(* CODESYS project FsGenerics_0.1.1.1.library
   Company: FisoThemes
   DefaultNamespace: FsGenerics
   Version: 0.1.1.1
   Placeholder: FsGenerics
   Author: Goodwill Mzumala
   Description: A library for handling generic data.
   Title: FsGenerics

Project tree, tasks and I/O mapping:
  libraries: FsCommon, * (FisoThemes); FsError, * (FisoThemes); Tc2_Standard, * (Beckhoff Automation GmbH); Tc2_System, * (Beckhoff Automation GmbH); Tc2_Utilities, * (Beckhoff Automation GmbH); Tc3_Module, * (Beckhoff Automation GmbH)
  DUTs/
  GVLs/
  ITFs/
  PARAMs/
  POUs/
    function F_AllocateMemoryGeneric [ST]
    function F_AnyToGeneric [ST]
    function F_AnyToString [ST]
    function F_CloneGeneric [ST]
    function F_CompareAny [ST]
    function F_CompareGenerics [ST]
    function F_CopyGeneric [ST]
    function F_DeallocateGeneric [ST]
    function F_GenericToDateTime [ST]
    function F_GenericToNumber [ST]
    function F_GenericToString [ST]
    function F_GenericToTime [ST]
    function F_GenericToTimeOfDay [ST]
    function F_IsBooleanGeneric [ST]
    function F_IsDateGeneric [ST]
    function F_IsIntegerGeneric [ST]
    function F_IsMatchingGenerics [ST]
    function F_IsNumberGeneric [ST]
    function F_IsPrimitiveGeneric [ST]
    function F_IsRealNumberGeneric [ST]
    function F_IsSignedIntegerGeneric [ST]
    function F_IsStringConvertableGeneric [ST]
    function F_IsStringGeneric [ST]
    function F_IsTimeGeneric [ST]
    function F_IsUnsignedIntegerGeneric [ST]
    function F_ResetGeneric [ST]
    function F_SwapAny [ST]
    function F_SwapGenericsParameters [ST]
    program PLAYGROUND [ST]
  Project Information/
    function F_GetCompany [ST]
    function F_GetTitle [ST]
    function F_GetVersion [ST]
  UMLs/
  Version/
    global variables Global_Version
  VISUs/
*)

// Version/Global_Version
{attribute 'TcGenerated'}
{attribute 'no-analysis'}
{attribute 'linkalways'}
// This function has been automatically generated from the project information.
VAR_GLOBAL CONSTANT
	{attribute 'const_non_replaced'}
	stLibVersion_FsGenerics : ST_LibVersion := (iMajor := 0, iMinor := 1, iBuild := 1, iRevision := 1, nFlags := 0, sVersion := '0.1.1.1');
END_VAR

// POUs/F_AllocateMemoryGeneric
// Allocates memory for an array of generic values.
// [warning] This function performs dynamic memory allocation. Ensure proper error handling
//           and resource management to avoid memory leaks or allocation failures.
FUNCTION F_AllocateMemoryGeneric : POINTER TO FsCommon.T_Generic // Pointer to the allocated memory for generic values.
VAR_INPUT
	Count : FsCommon.T_Size; // The number of `FsCommon.T_Generic` values to allocate memory for.
END_VAR
VAR_OUTPUT
	Error : FsError.T_Error; // Error information if memory allocation fails.
END_VAR
VAR
	i, End : FsCommon.T_Position;
END_VAR

IF Count = 0 THEN RETURN; END_IF

F_AllocateMemoryGeneric := FsCommon.F_AllocateMemory(Count * SIZEOF(FsCommon.T_Generic));

IF F_AllocateMemoryGeneric = 0 THEN 
	Error := FsError.F_CreateError(
		FsError.GVL_ErrorDescriptors.fbGeneralErrorCodes,
		FsError.E_GeneralErrorCode.ERR_MEMORY_ALLOCATION_FAILED);
	RETURN;
	END_IF

End := FsCommon.F_SizeToPosition(Count) - 1;
FOR i := 0 TO End DO
	F_AllocateMemoryGeneric[i].TypeClass := __SYSTEM.TYPE_CLASS.TYPE_NONE;
	END_FOR

END_FUNCTION

// POUs/F_AnyToGeneric
// Converts a value of any type to a generic type.
FUNCTION F_AnyToGeneric : FsCommon.T_Generic
VAR_INPUT
	Value : ANY; // The value to be converted to a generic type.
END_VAR

F_AnyToGeneric := Value;

END_FUNCTION

// POUs/F_AnyToString
// Converts a value of any type to its string representation.
FUNCTION F_AnyToString : Tc2_System.T_MaxString
VAR_INPUT
	Value : ANY; // The string representation of the value.
END_VAR
VAR_OUTPUT
	Error : FsError.T_Error; // Error information if the conversion fails.
END_VAR

F_AnyToString := F_GenericToString(Value, Error => Error);

END_FUNCTION

// POUs/F_GenericToString
// Converts a generic value to a string representation.
FUNCTION F_GenericToString : Tc2_System.T_MaxString // The string representation of the generic value.
VAR_INPUT
	Value : FsCommon.T_Generic; // The generic value to be converted to a string.
END_VAR
VAR_OUTPUT
	Error : FsError.T_Error; // Error information if the conversion fails.
END_VAR
VAR
	uValue : FsCommon.U_Pointer := (pVoid := Value.pValue);
END_VAR

IF uValue.pVoid = 0 THEN 
	Error := FsError.F_CreateError(
			FsError.GVL_ErrorDescriptors.fbGeneralErrorCodes,
			FsError.E_GeneralErrorCode.ERR_INVALID_POINTER);
	RETURN; 
	END_IF

CASE Value.TypeClass OF 
	__SYSTEM.TYPE_CLASS.TYPE_BOOL:
		F_GenericToString := TO_STRING(uValue.pBool^);
		
    __SYSTEM.TYPE_CLASS.TYPE_BYTE:
		F_GenericToString := TO_STRING(uValue.pByte^);
		
    __SYSTEM.TYPE_CLASS.TYPE_WORD:
		F_GenericToString := TO_STRING(uValue.pWord^);
		
    __SYSTEM.TYPE_CLASS.TYPE_DWORD:
		F_GenericToString := TO_STRING(uValue.pDWord^);
		
    __SYSTEM.TYPE_CLASS.TYPE_LWORD:
		F_GenericToString := TO_STRING(uValue.pLWord^);
		
    __SYSTEM.TYPE_CLASS.TYPE_SINT:
		F_GenericToString := TO_STRING(uValue.pSInt^);
		
    __SYSTEM.TYPE_CLASS.TYPE_INT:
		F_GenericToString := TO_STRING(uValue.pInt^);
		
    __SYSTEM.TYPE_CLASS.TYPE_DINT:
		F_GenericToString := TO_STRING(uValue.pDInt^);
		
    __SYSTEM.TYPE_CLASS.TYPE_LINT:
		F_GenericToString := TO_STRING(uValue.pLInt^);
		
    __SYSTEM.TYPE_CLASS.TYPE_USINT:
		F_GenericToString := TO_STRING(uValue.pUSInt^);
		
    __SYSTEM.TYPE_CLASS.TYPE_UINT:
		F_GenericToString := TO_STRING(uValue.pUInt^);
		
    __SYSTEM.TYPE_CLASS.TYPE_UDINT:
		F_GenericToString := TO_STRING(uValue.pUDInt^);
		
    __SYSTEM.TYPE_CLASS.TYPE_ULINT:
		F_GenericToString := TO_STRING(uValue.pULInt^);
		
   __SYSTEM.TYPE_CLASS.TYPE_REAL:
		F_GenericToString := TO_STRING(uValue.pReal^);
		
    __SYSTEM.TYPE_CLASS.TYPE_LREAL:
		F_GenericToString := TO_STRING(uValue.pLReal^);
		
    __SYSTEM.TYPE_CLASS.TYPE_STRING:
		Tc2_Utilities.STRNCPY(ADR(F_GenericToString),
							  uValue.pMaxString, 
							 SIZEOF(F_GenericToString));
		
   __SYSTEM.TYPE_CLASS.TYPE_WSTRING:
		Tc2_Utilities.WSTRING_TO_STRING2(ADR(F_GenericToString),
										 uValue.pMaxWString,
										 SIZEOF(F_GenericToString));
		
    __SYSTEM.TYPE_CLASS.TYPE_TIME:
		F_GenericToString := TO_STRING(uValue.pTime^);
		
    __SYSTEM.TYPE_CLASS.TYPE_DATE:
		F_GenericToString := TO_STRING(uValue.pDate^);
		
    __SYSTEM.TYPE_CLASS.TYPE_DATEANDTIME:
		F_GenericToString := TO_STRING(uValue.pDateAndTime^);
		
    __SYSTEM.TYPE_CLASS.TYPE_TIMEOFDAY:
		F_GenericToString := TO_STRING(uValue.pTimeOfDay^);
		
	__SYSTEM.TYPE_CLASS.TYPE_POINTER:
		F_GenericToString := TO_STRING(uValue.pNested^.pVoid);
		
	__SYSTEM.TYPE_CLASS.TYPE_LTIME:
		F_GenericToString := TO_STRING(uValue.pLTime^);
ELSE
	Error := FsError.F_CreateError(
			FsError.GVL_ErrorDescriptors.fbGeneralErrorCodes,
			FsError.E_GeneralErrorCode.ERR_TYPE_MISMATCH);
	END_CASE

END_FUNCTION

// POUs/F_CloneGeneric
// Clones a generic value by allocating memory and copying the contents.
// [warning] This function performs dynamic memory allocation. Ensure proper error handling
//           and resource management to avoid memory leaks or allocation failures.
// [note] Strings are only copied to their terminating characters.
FUNCTION F_CloneGeneric : FsCommon.T_Generic // The cloned generic value.
VAR_INPUT
	Value : FsCommon.T_Generic; // The generic value to be cloned.
END_VAR
VAR_OUTPUT
	Error : FsError.T_Error; // Error information if cloning fails.
END_VAR

IF Value.pValue = 0 OR_ELSE Value.diSize = 0 THEN 
	Error := FsError.F_CreateError(
			FsError.GVL_ErrorDescriptors.fbGeneralErrorCodes,
			FsError.E_GeneralErrorCode.ERR_INVALID_INPUT);
	F_CloneGeneric.diSize := 0;
	F_CloneGeneric.TypeClass := FsCommon.T_TypeClass.TYPE_NONE;
	RETURN; 
	END_IF

F_CloneGeneric.pValue := FsCommon.F_AllocateMemory(FsCommon.F_DintToSize(Value.diSize));

IF F_CloneGeneric.pValue = 0 THEN
	Error := FsError.F_CreateError(
		FsError.GVL_ErrorDescriptors.fbGeneralErrorCodes,
		FsError.E_GeneralErrorCode.ERR_MEMORY_ALLOCATION_FAILED);
	F_CloneGeneric.diSize := 0;
	F_CloneGeneric.TypeClass := __SYSTEM.TYPE_CLASS.TYPE_NONE;
	RETURN;
	END_IF
	
F_CloneGeneric.diSize := Value.diSize;
F_CloneGeneric.TypeClass := Value.TypeClass;
	
CASE Value.TypeClass OF
	__SYSTEM.TYPE_CLASS.TYPE_STRING:
		Tc2_Utilities.STRNCPY(
			F_CloneGeneric.pValue,
			Value.pValue,
			FsCommon.F_DintToSize(Value.diSize));
			
	__SYSTEM.TYPE_CLASS.TYPE_WSTRING:
		Tc2_Utilities.WSTRNCPY(
			F_CloneGeneric.pValue,
			Value.pValue,
			FsCommon.F_DintToSize(Value.diSize));
ELSE
	Tc2_System.MEMCPY(F_CloneGeneric.pValue, Value.pValue, FsCommon.F_DintToSize(Value.diSize));
	END_CASE

END_FUNCTION

// POUs/F_CompareAny
// Compares two values of any type and returns the result of the comparison.
// [note] This function will always return a result. If the types are not directly comparable
//        or if there is any ambiguity in the comparison, the `bIsAmbiguous` flag will be set to `TRUE`.
FUNCTION F_CompareAny : FsCommon.E_Comparison // The result of the comparison.
VAR_INPUT
	A : ANY; // Value to compare to B.
	B : ANY; // Value to compare to A.
END_VAR
VAR_OUTPUT
	// If TRUE, the comparison was performed, but the result is ambiguous or unreliable.
	// This can occur if the types of A and B are not directly comparable, or if the comparison logic does not support the specific types provided.
	bIsAmbiguous : BOOL;
END_VAR

F_CompareAny := F_CompareGenerics(A, B, bIsAmbiguous => bIsAmbiguous);

END_FUNCTION

// POUs/F_CompareGenerics
// Compares two generic values and returns the result of the comparison.
// [note] This function will always return a result. If the types are not directly comparable
//        or if there is any ambiguity in the comparison, the `bIsAmbiguous` flag will be set to `TRUE`.
FUNCTION F_CompareGenerics : FsCommon.E_Comparison // The result of the comparison.
VAR_INPUT
	A : FsCommon.T_Generic; // Generic value to compare to B.
	B : FsCommon.T_Generic; // Generic value to compare to A.
END_VAR
VAR_OUTPUT
	// If TRUE, the comparison was performed, but the result is ambiguous or unreliable.
	// This can occur if the types of A and B are not directly comparable, or if the comparison logic does not support the specific types provided.
	bIsAmbiguous : BOOL;
END_VAR
VAR
	uA, uB : FsCommon.U_Primitive;
END_VAR

IF F_IsNumberGeneric(A) AND_THEN F_IsNumberGeneric(B) THEN
	uA.fLReal := F_GenericToNumber(A);
	uB.fLReal := F_GenericToNumber(B);
	F_CompareGenerics := SEL(uA.fLReal = uB.fLReal,
							 SEL(uA.fLReal > uB.fLReal, FsCommon.E_Comparison.Less, FsCommon.E_Comparison.Greater),
							 FsCommon.E_Comparison.Equal);
	RETURN;
	END_IF
	
IF F_IsTimeGeneric(A) AND_THEN F_IsTimeGeneric(B) THEN
	uA.tLTime := F_GenericToTime(A);
	uB.tLTime := F_GenericToTime(B);
	F_CompareGenerics := SEL(uA.tLTime = uB.tLTime , 
							 SEL(uA.tLTime > uB.tLTime, FsCommon.E_Comparison.Less, FsCommon.E_Comparison.Greater),
							 FsCommon.E_Comparison.Equal);
	RETURN;
	END_IF

IF F_IsDateGeneric(A) AND_THEN F_IsDateGeneric(B) THEN
	uA.dtDateAndTime := F_GenericToDateTime(A);
	uB.dtDateAndTime := F_GenericToDateTime(B);
	F_CompareGenerics := SEL(uA.dtDateAndTime = uB.dtDateAndTime, 
							 SEL(uA.dtDateAndTime > uB.dtDateAndTime, FsCommon.E_Comparison.Less, FsCommon.E_Comparison.Greater),
							 FsCommon.E_Comparison.Equal);
	RETURN;
	END_IF

IF F_IsMatchingGenerics(A, B) THEN
	bIsAmbiguous := A.TypeClass = __SYSTEM.TYPE_CLASS.TYPE_USERDEF;
	
	A.diSize := SEL(A.TypeClass = __SYSTEM.TYPE_CLASS.TYPE_STRING, 
					SEL(A.TypeClass = __SYSTEM.TYPE_CLASS.TYPE_WSTRING, A.diSize, TO_DINT(Tc2_Utilities.WLEN2(A.pValue))),
					TO_DINT(Tc2_Utilities.LEN2(A.pValue)));
					
	B.diSize := SEL(B.TypeClass = __SYSTEM.TYPE_CLASS.TYPE_STRING,
					SEL(B.TypeClass = __SYSTEM.TYPE_CLASS.TYPE_WSTRING, B.diSize, TO_DINT(Tc2_Utilities.WLEN2(B.pValue))),
					TO_DINT(Tc2_Utilities.LEN2(B.pValue)));
					
	CASE Tc2_System.MEMCMP(A.pValue, B.pValue, TO_UDINT(MIN(A.diSize, B.diSize))) OF
		-1		: F_CompareGenerics := FsCommon.E_Comparison.Less;
		0		: F_CompareGenerics := FsCommon.E_Comparison.Equal;
		1		: F_CompareGenerics := FsCommon.E_Comparison.Greater;
		16#FF	:
			bIsAmbiguous := TRUE; 
			F_CompareGenerics := SEL(A.diSize = B.diSize,
									 SEL(A.diSize > B.diSize, FsCommon.E_Comparison.Less, FsCommon.E_Comparison.Greater),
									 FsCommon.E_Comparison.Equal);
		END_CASE
	RETURN;
	END_IF
	
bIsAmbiguous := TRUE;
F_CompareGenerics := SEL(A.TypeClass > B.TypeClass, FsCommon.E_Comparison.Less, FsCommon.E_Comparison.Greater);

END_FUNCTION

// POUs/F_IsNumberGeneric
// Checks if the given generic value represents a numeric type.
FUNCTION F_IsNumberGeneric : BOOL // TRUE if the generic value represents a numeric type.
VAR_INPUT
	Value : FsCommon.T_Generic; // The generic value to check.
END_VAR

CASE Value.TypeClass OF
	__SYSTEM.TYPE_CLASS.TYPE_BYTE,
	__SYSTEM.TYPE_CLASS.TYPE_WORD,
	__SYSTEM.TYPE_CLASS.TYPE_DWORD,
	__SYSTEM.TYPE_CLASS.TYPE_LWORD,
	__SYSTEM.TYPE_CLASS.TYPE_SINT,
	__SYSTEM.TYPE_CLASS.TYPE_INT,
	__SYSTEM.TYPE_CLASS.TYPE_DINT,
	__SYSTEM.TYPE_CLASS.TYPE_LINT,
	__SYSTEM.TYPE_CLASS.TYPE_USINT,
	__SYSTEM.TYPE_CLASS.TYPE_UINT,
	__SYSTEM.TYPE_CLASS.TYPE_UDINT,
	__SYSTEM.TYPE_CLASS.TYPE_ULINT,
	__SYSTEM.TYPE_CLASS.TYPE_REAL,
	__SYSTEM.TYPE_CLASS.TYPE_LREAL,
	__SYSTEM.TYPE_CLASS.TYPE_POINTER:
		F_IsNumberGeneric := TRUE;
	END_CASE

END_FUNCTION

// POUs/F_GenericToNumber
// Converts a generic value to an LREAL (floating-point number) based on its type class.
FUNCTION F_GenericToNumber : LREAL // The converted floating-point number.
VAR_INPUT
	Value : FsCommon.T_Generic; // The generic value to convert to LREAL.
END_VAR
VAR_OUTPUT
	Error : FsError.T_Error; // Error information if the conversion fails.
END_VAR
VAR
	uValue : FsCommon.U_Pointer := (pVoid := Value.pValue);
END_VAR

IF uValue.pVoid = 0 THEN 
	Error := FsError.F_CreateError(
			FsError.GVL_ErrorDescriptors.fbGeneralErrorCodes,
			FsError.E_GeneralErrorCode.ERR_INVALID_POINTER);
	RETURN; 
	END_IF

CASE Value.TypeClass OF 
	__SYSTEM.TYPE_CLASS.TYPE_BOOL:
		F_GenericToNumber := TO_LREAL(uValue.pBool^);
		
    __SYSTEM.TYPE_CLASS.TYPE_BYTE:
		F_GenericToNumber := TO_LREAL(uValue.pByte^);
		
    __SYSTEM.TYPE_CLASS.TYPE_WORD:
		F_GenericToNumber := TO_LREAL(uValue.pWord^);
		
    __SYSTEM.TYPE_CLASS.TYPE_DWORD:
		F_GenericToNumber := TO_LREAL(uValue.pDWord^);
		
    __SYSTEM.TYPE_CLASS.TYPE_LWORD:
		F_GenericToNumber := TO_LREAL(uValue.pLWord^);
		
    __SYSTEM.TYPE_CLASS.TYPE_SINT:
		F_GenericToNumber := TO_LREAL(uValue.pSInt^);
		
    __SYSTEM.TYPE_CLASS.TYPE_INT:
		F_GenericToNumber := TO_LREAL(uValue.pInt^);
		
    __SYSTEM.TYPE_CLASS.TYPE_DINT:
		F_GenericToNumber := TO_LREAL(uValue.pDInt^);
		
    __SYSTEM.TYPE_CLASS.TYPE_LINT:
		F_GenericToNumber := TO_LREAL(uValue.pLInt^);
		
    __SYSTEM.TYPE_CLASS.TYPE_USINT:
		F_GenericToNumber := TO_LREAL(uValue.pUSInt^);
		
    __SYSTEM.TYPE_CLASS.TYPE_UINT:
		F_GenericToNumber := TO_LREAL(uValue.pUInt^);
		
    __SYSTEM.TYPE_CLASS.TYPE_UDINT:
		F_GenericToNumber := TO_LREAL(uValue.pUDInt^);
		
    __SYSTEM.TYPE_CLASS.TYPE_ULINT:
		F_GenericToNumber := TO_LREAL(uValue.pULInt^);
		
   __SYSTEM.TYPE_CLASS.TYPE_REAL:
		F_GenericToNumber := TO_LREAL(uValue.pReal^);
		
    __SYSTEM.TYPE_CLASS.TYPE_LREAL:
		F_GenericToNumber := TO_LREAL(uValue.pLReal^);
		
    __SYSTEM.TYPE_CLASS.TYPE_STRING:
		F_GenericToNumber := TO_LREAL(uValue.pString^);
		
   __SYSTEM.TYPE_CLASS.TYPE_WSTRING:
		F_GenericToNumber := TO_LREAL(uValue.pWString^);
		
    __SYSTEM.TYPE_CLASS.TYPE_TIME:
		F_GenericToNumber := TO_LREAL(uValue.pTime^);
		
    __SYSTEM.TYPE_CLASS.TYPE_DATE:
		F_GenericToNumber := TO_LREAL(uValue.pDate^);
		
    __SYSTEM.TYPE_CLASS.TYPE_DATEANDTIME:
		F_GenericToNumber := TO_LREAL(uValue.pDateAndTime^);

    __SYSTEM.TYPE_CLASS.TYPE_TIMEOFDAY:
		F_GenericToNumber := TO_LREAL(uValue.pTimeOfDay^);
		
	__SYSTEM.TYPE_CLASS.TYPE_POINTER:
		F_GenericToNumber := TO_LREAL(uValue.pNested^.pVoid);
		
	__SYSTEM.TYPE_CLASS.TYPE_LTIME:
		F_GenericToNumber := TO_LREAL(uValue.pLTime^);
ELSE
	Error := FsError.F_CreateError(
			FsError.GVL_ErrorDescriptors.fbGeneralErrorCodes,
			FsError.E_GeneralErrorCode.ERR_TYPE_MISMATCH);
	END_CASE

END_FUNCTION

// POUs/F_IsTimeGeneric
// Checks if the given generic value is of time-related type.
FUNCTION F_IsTimeGeneric : BOOL // TRUE if the generic value is a time-related type.
VAR_INPUT
	Value : FsCommon.T_Generic; // The generic value to check.
END_VAR

CASE Value.TypeClass OF
	__SYSTEM.TYPE_CLASS.TYPE_TIME,
	__SYSTEM.TYPE_CLASS.TYPE_LTIME,
	__SYSTEM.TYPE_CLASS.TYPE_DATEANDTIME,
	__SYSTEM.TYPE_CLASS.TYPE_TIMEOFDAY:
		F_IsTimeGeneric := TRUE;
	END_CASE

END_FUNCTION

// POUs/F_GenericToTime
// Converts a generic value to LTIME based on its type class.
FUNCTION F_GenericToTime : LTIME // The converted LTIME value.
VAR_INPUT
	Value : FsCommon.T_Generic; // The generic value to convert to LTIME.
END_VAR
VAR_OUTPUT
	Error : FsError.T_Error; // Error information if the conversion fails.
END_VAR
VAR
	uValue : FsCommon.U_Pointer := (pVoid := Value.pValue);
END_VAR

IF uValue.pVoid = 0 THEN 
	Error := FsError.F_CreateError(
			FsError.GVL_ErrorDescriptors.fbGeneralErrorCodes,
			FsError.E_GeneralErrorCode.ERR_INVALID_POINTER);
	RETURN; 
	END_IF

CASE Value.TypeClass OF 
	__SYSTEM.TYPE_CLASS.TYPE_BOOL:
		F_GenericToTime := TO_LTIME(uValue.pBool^);
		
    __SYSTEM.TYPE_CLASS.TYPE_BYTE:
		F_GenericToTime := TO_LTIME(uValue.pByte^);
		
    __SYSTEM.TYPE_CLASS.TYPE_WORD:
		F_GenericToTime := TO_LTIME(uValue.pWord^);
		
    __SYSTEM.TYPE_CLASS.TYPE_DWORD:
		F_GenericToTime := TO_LTIME(uValue.pDWord^);
		
    __SYSTEM.TYPE_CLASS.TYPE_LWORD:
		F_GenericToTime := TO_LTIME(uValue.pLWord^);
		
    __SYSTEM.TYPE_CLASS.TYPE_SINT:
		F_GenericToTime := TO_LTIME(uValue.pSInt^);
		
    __SYSTEM.TYPE_CLASS.TYPE_INT:
		F_GenericToTime := TO_LTIME(uValue.pInt^);
		
    __SYSTEM.TYPE_CLASS.TYPE_DINT:
		F_GenericToTime := TO_LTIME(uValue.pDInt^);
		
    __SYSTEM.TYPE_CLASS.TYPE_LINT:
		F_GenericToTime := TO_LTIME(uValue.pLInt^);
		
    __SYSTEM.TYPE_CLASS.TYPE_USINT:
		F_GenericToTime := TO_LTIME(uValue.pUSInt^);
		
    __SYSTEM.TYPE_CLASS.TYPE_UINT:
		F_GenericToTime := TO_LTIME(uValue.pUInt^);
		
    __SYSTEM.TYPE_CLASS.TYPE_UDINT:
		F_GenericToTime := TO_LTIME(uValue.pUDInt^);
		
    __SYSTEM.TYPE_CLASS.TYPE_ULINT:
		F_GenericToTime := TO_LTIME(uValue.pULInt^);
		
   __SYSTEM.TYPE_CLASS.TYPE_REAL:
		F_GenericToTime := TO_LTIME(uValue.pReal^);
		
    __SYSTEM.TYPE_CLASS.TYPE_LREAL:
		F_GenericToTime := TO_LTIME(uValue.pLReal^);
		
    __SYSTEM.TYPE_CLASS.TYPE_STRING:
		F_GenericToTime := TO_LTIME(uValue.pString^);
		
   __SYSTEM.TYPE_CLASS.TYPE_WSTRING:
		F_GenericToTime := TO_LTIME(uValue.pWString^);
		
    __SYSTEM.TYPE_CLASS.TYPE_TIME:
		F_GenericToTime := TO_LTIME(uValue.pTime^);
		
    __SYSTEM.TYPE_CLASS.TYPE_DATE:
		F_GenericToTime := TO_LTIME(uValue.pDate^);
		
    __SYSTEM.TYPE_CLASS.TYPE_DATEANDTIME:
		F_GenericToTime := TO_LTIME(uValue.pDateAndTime^);
		
    __SYSTEM.TYPE_CLASS.TYPE_TIMEOFDAY:
		F_GenericToTime := TO_LTIME(uValue.pTimeOfDay^);
		
	__SYSTEM.TYPE_CLASS.TYPE_LTIME:
		F_GenericToTime := uValue.pLTime^;
ELSE
	Error := FsError.F_CreateError(
			FsError.GVL_ErrorDescriptors.fbGeneralErrorCodes,
			FsError.E_GeneralErrorCode.ERR_TYPE_MISMATCH);
	END_CASE

END_FUNCTION

// POUs/F_IsDateGeneric
// Checks if the given generic value is of date or date and time type.
FUNCTION F_IsDateGeneric : BOOL // TRUE if the generic value is date or date and time.
VAR_INPUT
	Value : FsCommon.T_Generic; // The generic value to check.
END_VAR

F_IsDateGeneric := 
	Value.TypeClass = __SYSTEM.TYPE_CLASS.TYPE_DATE 
	OR 
	Value.TypeClass = __SYSTEM.TYPE_CLASS.TYPE_DATEANDTIME;

END_FUNCTION

// POUs/F_GenericToDateTime
// Converts a generic value to a DT (DateTime) type based on its type class.
// [note] This function handles different types and performs the conversion accordingly.
//        If the type of the generic value is not supported for conversion to DT, 
//        an error will be returned.
FUNCTION F_GenericToDateTime : DT // The converted DateTime value.
VAR_INPUT
	Value : FsCommon.T_Generic; // The generic value to convert to DateTime.
END_VAR
VAR_OUTPUT
	Error : FsError.T_Error; // Error information if the conversion fails.
END_VAR
VAR
	uValue : FsCommon.U_Pointer := (pVoid := Value.pValue);
END_VAR

IF uValue.pVoid = 0 THEN 
	Error := FsError.F_CreateError(
			FsError.GVL_ErrorDescriptors.fbGeneralErrorCodes,
			FsError.E_GeneralErrorCode.ERR_INVALID_POINTER);
	RETURN; 
	END_IF

CASE Value.TypeClass OF 
	__SYSTEM.TYPE_CLASS.TYPE_BOOL:
		F_GenericToDateTime := TO_DT(uValue.pBool^);
		
    __SYSTEM.TYPE_CLASS.TYPE_BYTE:
		F_GenericToDateTime := TO_DT(uValue.pByte^);
		
    __SYSTEM.TYPE_CLASS.TYPE_WORD:
		F_GenericToDateTime := TO_DT(uValue.pWord^);
		
    __SYSTEM.TYPE_CLASS.TYPE_DWORD:
		F_GenericToDateTime := TO_DT(uValue.pDWord^);
		
    __SYSTEM.TYPE_CLASS.TYPE_LWORD:
		F_GenericToDateTime := TO_DT(uValue.pLWord^);
		
    __SYSTEM.TYPE_CLASS.TYPE_SINT:
		F_GenericToDateTime := TO_DT(uValue.pSInt^);
		
    __SYSTEM.TYPE_CLASS.TYPE_INT:
		F_GenericToDateTime := TO_DT(uValue.pInt^);
		
    __SYSTEM.TYPE_CLASS.TYPE_DINT:
		F_GenericToDateTime := TO_DT(uValue.pDInt^);
		
    __SYSTEM.TYPE_CLASS.TYPE_LINT:
		F_GenericToDateTime := TO_DT(uValue.pLInt^);
		
    __SYSTEM.TYPE_CLASS.TYPE_USINT:
		F_GenericToDateTime := TO_DT(uValue.pUSInt^);
		
    __SYSTEM.TYPE_CLASS.TYPE_UINT:
		F_GenericToDateTime := TO_DT(uValue.pUInt^);
		
    __SYSTEM.TYPE_CLASS.TYPE_UDINT:
		F_GenericToDateTime := TO_DT(uValue.pUDInt^);
		
    __SYSTEM.TYPE_CLASS.TYPE_ULINT:
		F_GenericToDateTime := TO_DT(uValue.pULInt^);
		
   __SYSTEM.TYPE_CLASS.TYPE_REAL:
		F_GenericToDateTime := TO_DT(uValue.pReal^);
		
    __SYSTEM.TYPE_CLASS.TYPE_LREAL:
		F_GenericToDateTime := TO_DT(uValue.pLReal^);
		
    __SYSTEM.TYPE_CLASS.TYPE_STRING:
		F_GenericToDateTime := TO_DT(uValue.pString^);
		
   __SYSTEM.TYPE_CLASS.TYPE_WSTRING:
		F_GenericToDateTime := TO_DT(uValue.pWString^);
		
    __SYSTEM.TYPE_CLASS.TYPE_TIME:
		F_GenericToDateTime := TO_DT(uValue.pTime^);
		
    __SYSTEM.TYPE_CLASS.TYPE_DATE:
		F_GenericToDateTime := TO_DT(uValue.pDate^);
		
    __SYSTEM.TYPE_CLASS.TYPE_DATEANDTIME:
		F_GenericToDateTime := TO_DT(uValue.pDateAndTime^);
		
    __SYSTEM.TYPE_CLASS.TYPE_TIMEOFDAY:
		F_GenericToDateTime := TO_DT(uValue.pTimeOfDay^);
		
	__SYSTEM.TYPE_CLASS.TYPE_LTIME:
		F_GenericToDateTime := TO_DT(uValue.pLTime^);
ELSE
	Error := FsError.F_CreateError(
			FsError.GVL_ErrorDescriptors.fbGeneralErrorCodes,
			FsError.E_GeneralErrorCode.ERR_TYPE_MISMATCH);
	END_CASE

END_FUNCTION

// POUs/F_IsMatchingGenerics
// Checks if two generic values match in type and size.
// [note] For string types only their types are compared.
FUNCTION F_IsMatchingGenerics : BOOL // TRUE if the generic values match in type and size (size is only for none string types).
VAR_INPUT
	A : FsCommon.T_Generic; // Generic value to compare with B.
	B : FsCommon.T_Generic; // Generic value to compare with A.
END_VAR

CASE A.TypeClass OF 
	__SYSTEM.TYPE_CLASS.TYPE_STRING,
	__SYSTEM.TYPE_CLASS.TYPE_WSTRING: 
		F_IsMatchingGenerics := A.TypeClass = B.TypeClass;
ELSE
	F_IsMatchingGenerics := A.diSize = B.diSize AND A.TypeClass = B.TypeClass;
	END_CASE

END_FUNCTION

// POUs/F_CopyGeneric
// Copies data from the source generic value to the destination generic value.
FUNCTION F_CopyGeneric
VAR_IN_OUT
	Source 		: FsCommon.T_Generic; // The source generic value from which data will be copied.
	Destination : FsCommon.T_Generic; // The destination generic value to which data will be copied.
END_VAR
VAR_OUTPUT
	Error : FsError.T_Error; // Error information if copying fails.
END_VAR

IF Source.diSize <> Destination.diSize THEN 
	Error := FsError.F_CreateError(
			FsError.GVL_ErrorDescriptors.fbGeneralErrorCodes,
			FsError.E_GeneralErrorCode.ERR_SIZE_MISMATCH);
	RETURN; 
	END_IF
	
IF Source.pValue = 0 OR Destination.pValue = 0 THEN 
	Error := FsError.F_CreateError(
			FsError.GVL_ErrorDescriptors.fbGeneralErrorCodes,
			FsError.E_GeneralErrorCode.ERR_INVALID_POINTER);
	RETURN; 
	END_IF
	
Tc2_System.MEMCPY(
	Destination.pValue,
	Source.pValue,
	FsCommon.F_DintToSize(Destination.diSize));

END_FUNCTION

// POUs/F_DeallocateGeneric
// Deallocates memory associated with a generic value and resets it to a default state.
FUNCTION F_DeallocateGeneric
VAR_IN_OUT
	Value : FsCommon.T_Generic; // The generic value whose memory will be deallocated.
END_VAR

FsCommon.F_DeallocateMemory(Value.pValue);
Value.diSize := 0;
Value.TypeClass := __SYSTEM.TYPE_CLASS.TYPE_NONE;

END_FUNCTION

// POUs/F_GenericToTimeOfDay
// Converts a generic value to TOD (Time of Day) based on its type class.
FUNCTION F_GenericToTimeOfDay : TOD // The converted TOD value.
VAR_INPUT
	Value : FsCommon.T_Generic; // The generic value to convert to TOD.
END_VAR
VAR_OUTPUT
	Error : FsError.T_Error; // Error information if conversion fails.
END_VAR
VAR
	uValue : FsCommon.U_Pointer := (pVoid := Value.pValue);
END_VAR

IF uValue.pVoid = 0 THEN 
	Error := FsError.F_CreateError(
			FsError.GVL_ErrorDescriptors.fbGeneralErrorCodes,
			FsError.E_GeneralErrorCode.ERR_INVALID_POINTER);
	RETURN; 
	END_IF

CASE Value.TypeClass OF 
	__SYSTEM.TYPE_CLASS.TYPE_BOOL:
		F_GenericToTimeOfDay := TO_TOD(uValue.pBool^);
		
    __SYSTEM.TYPE_CLASS.TYPE_BYTE:
		F_GenericToTimeOfDay := TO_TOD(uValue.pByte^);
		
    __SYSTEM.TYPE_CLASS.TYPE_WORD:
		F_GenericToTimeOfDay := TO_TOD(uValue.pWord^);
		
    __SYSTEM.TYPE_CLASS.TYPE_DWORD:
		F_GenericToTimeOfDay := TO_TOD(uValue.pDWord^);
		
    __SYSTEM.TYPE_CLASS.TYPE_LWORD:
		F_GenericToTimeOfDay := TO_TOD(uValue.pLWord^);
		
    __SYSTEM.TYPE_CLASS.TYPE_SINT:
		F_GenericToTimeOfDay := TO_TOD(uValue.pSint^);
		
    __SYSTEM.TYPE_CLASS.TYPE_INT:
		F_GenericToTimeOfDay := TO_TOD(uValue.pInt^);
		
    __SYSTEM.TYPE_CLASS.TYPE_DINT:
		F_GenericToTimeOfDay := TO_TOD(uValue.pDint^);
		
    __SYSTEM.TYPE_CLASS.TYPE_LINT:
		F_GenericToTimeOfDay := TO_TOD(uValue.pLint^);
		
    __SYSTEM.TYPE_CLASS.TYPE_USINT:
		F_GenericToTimeOfDay := TO_TOD(uValue.pUSint^);
		
    __SYSTEM.TYPE_CLASS.TYPE_UINT:
		F_GenericToTimeOfDay := TO_TOD(uValue.pUInt^);
		
    __SYSTEM.TYPE_CLASS.TYPE_UDINT:
		F_GenericToTimeOfDay := TO_TOD(uValue.pUDint^);
		
    __SYSTEM.TYPE_CLASS.TYPE_ULINT:
		F_GenericToTimeOfDay := TO_TOD(uValue.pULint^);
		
   __SYSTEM.TYPE_CLASS.TYPE_REAL:
		F_GenericToTimeOfDay := TO_TOD(uValue.pReal^);
		
    __SYSTEM.TYPE_CLASS.TYPE_LREAL:
		F_GenericToTimeOfDay := TO_TOD(uValue.pLReal^);
		
    __SYSTEM.TYPE_CLASS.TYPE_STRING:
		F_GenericToTimeOfDay := TO_TOD(uValue.pString^);
		
   __SYSTEM.TYPE_CLASS.TYPE_WSTRING:
		F_GenericToTimeOfDay := TO_TOD(uValue.pWString^);
		
    __SYSTEM.TYPE_CLASS.TYPE_TIME:
		F_GenericToTimeOfDay := TO_TOD(uValue.pTime^);
		
    __SYSTEM.TYPE_CLASS.TYPE_DATE:
		F_GenericToTimeOfDay := TO_TOD(uValue.pDate^);
		
    __SYSTEM.TYPE_CLASS.TYPE_DATEANDTIME:
		F_GenericToTimeOfDay := TO_TOD(uValue.pDateAndTime^);
		
    __SYSTEM.TYPE_CLASS.TYPE_TIMEOFDAY:
		F_GenericToTimeOfDay := uValue.pTimeOfDay^;
		
	__SYSTEM.TYPE_CLASS.TYPE_LTIME:
		F_GenericToTimeOfDay := TO_TOD(uValue.pLTime^);
ELSE
	Error := FsError.F_CreateError(
			FsError.GVL_ErrorDescriptors.fbGeneralErrorCodes,
			FsError.E_GeneralErrorCode.ERR_TYPE_MISMATCH);
	END_CASE

END_FUNCTION

// POUs/F_IsBooleanGeneric
// Checks if the given generic value is of boolean type.
FUNCTION F_IsBooleanGeneric : BOOL // TRUE if the generic value is boolean.
VAR_INPUT
	Value : FsCommon.T_Generic; // The generic value to check.
END_VAR

F_IsBooleanGeneric := Value.TypeClass = __SYSTEM.TYPE_CLASS.TYPE_BOOL;

END_FUNCTION

// POUs/F_IsIntegerGeneric
// Checks if the given generic value is of integer type.
FUNCTION F_IsIntegerGeneric : BOOL // TRUE if the generic value is integer.
VAR_INPUT
	Value : FsCommon.T_Generic; // The generic value to check.
END_VAR

CASE Value.TypeClass OF
	__SYSTEM.TYPE_CLASS.TYPE_BYTE,
	__SYSTEM.TYPE_CLASS.TYPE_WORD,
	__SYSTEM.TYPE_CLASS.TYPE_DWORD,
	__SYSTEM.TYPE_CLASS.TYPE_LWORD,
	__SYSTEM.TYPE_CLASS.TYPE_SINT,
	__SYSTEM.TYPE_CLASS.TYPE_INT,
	__SYSTEM.TYPE_CLASS.TYPE_DINT,
	__SYSTEM.TYPE_CLASS.TYPE_LINT,
	__SYSTEM.TYPE_CLASS.TYPE_USINT,
	__SYSTEM.TYPE_CLASS.TYPE_UINT,
	__SYSTEM.TYPE_CLASS.TYPE_UDINT,
	__SYSTEM.TYPE_CLASS.TYPE_ULINT:
		F_IsIntegerGeneric := TRUE;
	END_CASE

END_FUNCTION

// POUs/F_IsPrimitiveGeneric
// Checks if the given generic value represents a primitive type.
FUNCTION F_IsPrimitiveGeneric : BOOL // TRUE if the generic value represents a primitive type, FALSE otherwise.
VAR_INPUT
	Value : FsCommon.T_Generic; // The generic value to check.
END_VAR

CASE Value.TypeClass OF
	__SYSTEM.TYPE_CLASS.TYPE_BOOL,
	__SYSTEM.TYPE_CLASS.TYPE_BYTE,
	__SYSTEM.TYPE_CLASS.TYPE_WORD,
	__SYSTEM.TYPE_CLASS.TYPE_DWORD,
	__SYSTEM.TYPE_CLASS.TYPE_LWORD,
	__SYSTEM.TYPE_CLASS.TYPE_SINT,
	__SYSTEM.TYPE_CLASS.TYPE_INT,
	__SYSTEM.TYPE_CLASS.TYPE_DINT,
	__SYSTEM.TYPE_CLASS.TYPE_LINT,
	__SYSTEM.TYPE_CLASS.TYPE_USINT,
	__SYSTEM.TYPE_CLASS.TYPE_UINT,
	__SYSTEM.TYPE_CLASS.TYPE_UDINT,
	__SYSTEM.TYPE_CLASS.TYPE_ULINT,
	__SYSTEM.TYPE_CLASS.TYPE_REAL,
	__SYSTEM.TYPE_CLASS.TYPE_LREAL,
	__SYSTEM.TYPE_CLASS.TYPE_TIME,
	__SYSTEM.TYPE_CLASS.TYPE_LTIME,
	__SYSTEM.TYPE_CLASS.TYPE_DATE,
	__SYSTEM.TYPE_CLASS.TYPE_DATEANDTIME,
	__SYSTEM.TYPE_CLASS.TYPE_TIMEOFDAY,
	__SYSTEM.TYPE_CLASS.TYPE_POINTER:
		F_IsPrimitiveGeneric := TRUE;
	END_CASE

END_FUNCTION

// POUs/F_IsRealNumberGeneric
// Checks if the given generic value represents a real (floating-point) number type.
FUNCTION F_IsRealNumberGeneric : BOOL // TRUE if the generic value represents a real (floating-point) number type.
VAR_INPUT
	Value : FsCommon.T_Generic; // The generic value to check.
END_VAR

F_IsRealNumberGeneric := 
	Value.TypeClass = __SYSTEM.TYPE_CLASS.TYPE_REAL
	OR
	Value.TypeClass = __SYSTEM.TYPE_CLASS.TYPE_LREAL;

END_FUNCTION

// POUs/F_IsSignedIntegerGeneric
// Checks if the given generic value represents a signed integer type.
FUNCTION F_IsSignedIntegerGeneric : BOOL // TRUE if the generic value represents a signed integer type.
VAR_INPUT
	Value : FsCommon.T_Generic; // The generic value to check.
END_VAR

CASE Value.TypeClass OF
	__SYSTEM.TYPE_CLASS.TYPE_SINT,
	__SYSTEM.TYPE_CLASS.TYPE_INT,
	__SYSTEM.TYPE_CLASS.TYPE_DINT,
	__SYSTEM.TYPE_CLASS.TYPE_LINT:
		F_IsSignedIntegerGeneric := TRUE;
	END_CASE

END_FUNCTION

// POUs/F_IsStringConvertableGeneric
// Checks if the given generic value can be converted to a string type.
FUNCTION F_IsStringConvertableGeneric : BOOL // TRUE if the generic value can be converted to a string type.
VAR_INPUT
	Value : FsCommon.T_Generic; // The generic value to check.
END_VAR

CASE Value.TypeClass OF
	__SYSTEM.TYPE_CLASS.TYPE_STRING,
	__SYSTEM.TYPE_CLASS.TYPE_WSTRING,
	__SYSTEM.TYPE_CLASS.TYPE_BOOL,
	__SYSTEM.TYPE_CLASS.TYPE_BYTE,
	__SYSTEM.TYPE_CLASS.TYPE_WORD,
	__SYSTEM.TYPE_CLASS.TYPE_DWORD,
	__SYSTEM.TYPE_CLASS.TYPE_LWORD,
	__SYSTEM.TYPE_CLASS.TYPE_SINT,
	__SYSTEM.TYPE_CLASS.TYPE_INT,
	__SYSTEM.TYPE_CLASS.TYPE_DINT,
	__SYSTEM.TYPE_CLASS.TYPE_LINT,
	__SYSTEM.TYPE_CLASS.TYPE_USINT,
	__SYSTEM.TYPE_CLASS.TYPE_UINT,
	__SYSTEM.TYPE_CLASS.TYPE_UDINT,
	__SYSTEM.TYPE_CLASS.TYPE_ULINT,
	__SYSTEM.TYPE_CLASS.TYPE_REAL,
	__SYSTEM.TYPE_CLASS.TYPE_LREAL,
	__SYSTEM.TYPE_CLASS.TYPE_TIME,
	__SYSTEM.TYPE_CLASS.TYPE_LTIME,
	__SYSTEM.TYPE_CLASS.TYPE_DATE,
	__SYSTEM.TYPE_CLASS.TYPE_DATEANDTIME,
	__SYSTEM.TYPE_CLASS.TYPE_TIMEOFDAY,
	__SYSTEM.TYPE_CLASS.TYPE_POINTER:
		F_IsStringConvertableGeneric := TRUE;
	END_CASE

END_FUNCTION

// POUs/F_IsStringGeneric
// Checks if the given generic value is of string type.
FUNCTION F_IsStringGeneric : BOOL // TRUE if the generic value is a string type.
VAR_INPUT
	Value : FsCommon.T_Generic; // The generic value to check.
END_VAR

F_IsStringGeneric := 
	Value.TypeClass = __SYSTEM.TYPE_CLASS.TYPE_STRING 
	OR 
	Value.TypeClass = __SYSTEM.TYPE_CLASS.TYPE_WSTRING;

END_FUNCTION

// POUs/F_IsUnsignedIntegerGeneric
// Checks if the given generic value is an unsigned integer type.
FUNCTION F_IsUnsignedIntegerGeneric : BOOL // TRUE if the generic value is an unsigned integer type.
VAR_INPUT
	Value : FsCommon.T_Generic; // The generic value to check.
END_VAR

CASE Value.TypeClass OF
	__SYSTEM.TYPE_CLASS.TYPE_BYTE,
	__SYSTEM.TYPE_CLASS.TYPE_WORD,
	__SYSTEM.TYPE_CLASS.TYPE_DWORD,
	__SYSTEM.TYPE_CLASS.TYPE_LWORD,
	__SYSTEM.TYPE_CLASS.TYPE_USINT,
	__SYSTEM.TYPE_CLASS.TYPE_UINT,
	__SYSTEM.TYPE_CLASS.TYPE_UDINT,
	__SYSTEM.TYPE_CLASS.TYPE_ULINT:
		F_IsUnsignedIntegerGeneric := TRUE;
	END_CASE

END_FUNCTION

// POUs/F_ResetGeneric
// Resets the content and type information of a generic value.
// [note] This function resets the internal state of the generic value 
//        by setting its pointer, size, and type class to default values. 
//        It does not deallocate or free any memory associated with the 
//        generic value.
FUNCTION F_ResetGeneric
VAR_IN_OUT
	Value : FsCommon.T_Generic; // The generic value to reset.
END_VAR

Value.pValue := 0;
Value.diSize := 0;
Value.TypeClass := __SYSTEM.TYPE_CLASS.TYPE_NONE;

END_FUNCTION

// POUs/F_SwapAny
// Swaps the contents of two variables of any type, assuming they are of the same type and size.
// [warning] This function only performs size checks and not type checks before swapping.
FUNCTION F_SwapAny
VAR_INPUT
    A : ANY; // Variable A to swap.
    B : ANY; // Variable B to swap.
END_VAR
VAR_OUTPUT
    Error : FsError.T_Error; // Error information if swapping fails.
END_VAR

IF A.diSize <> B.diSize THEN 
	Error := FsError.F_CreateError(FsError.GVL_ErrorDescriptors.fbGeneralErrorCodes,
								   FsError.E_GeneralErrorCode.ERR_SIZE_MISMATCH);
	RETURN;
	END_IF

FsCommon.F_SwapMemory(A.pValue, B.pValue, FsCommon.F_DintToSize(A.diSize));

END_FUNCTION

// POUs/F_SwapGenericsParameters
// Swaps the parameters of two generic values.
FUNCTION F_SwapGenericsParameters
VAR_IN_OUT
	A : FsCommon.T_Generic; // Generic whose parameters will be swapped with B.
	B : FsCommon.T_Generic; // Generic whose parameters will be swapped with B.
END_VAR
VAR
	Tmp : FsCommon.T_Generic;
END_VAR

Tmp := A;
A 	:= B;
B 	:= Tmp;

END_FUNCTION

// POUs/PLAYGROUND
{attribute 'no_explicit_call' := 'direct call for this program is not allowed'} 
PROGRAM INTERNAL PLAYGROUND
VAR
	t_Value : STRING;
	pValue : POINTER TO STRING := ADR(t_Value);
	eComp : FsCommon.E_Comparison;
	nVal0 : DT := DT#1970-1-1-0:0:24;
	nVal1 : DT := DT#1970-1-1-0:0:12;
	dtDateTime : DT;
	bStart : BOOL := TRUE;
	Value : FsCommon.T_Generic;
	Error : FsError.T_Error;
	fbWithAdsLogger : FsError.FB_AdsErrorLogger;
END_VAR

t_Value := F_GenericToString(F_AnyToGeneric(pValue));
eComp := F_CompareGenerics(F_AnyToGeneric(nVal0), F_AnyToGeneric(nVal1));

IF FsCommon.F_ResetOnTrue(bStart) THEN 
	F_SwapAny(nVal0 , nVal1, Error => Error); 
	IF Error.IsRaised THEN Error.LogMessage(fbWithAdsLogger); END_IF
	END_IF


(*
F_CloneGeneric(Value, Error => Error);
IF Error.IsRaised THEN 
	// Handle error.
	Error.LogMessage(fbWithAdsLogger);
	END_IF
	
*)

END_PROGRAM

// Project Information/F_GetCompany
// This function has been automatically generated from the project information.
{attribute 'signature_flag' := '1073741824'}
{attribute 'TcGenerated'}
{attribute 'no-analysis'}
FUNCTION F_GetCompany : WSTRING
VAR_INPUT
	
END_VAR

F_GetCompany := "FisoThemes";

END_FUNCTION

// Project Information/F_GetTitle
// This function has been automatically generated from the project information.
{attribute 'signature_flag' := '1073741824'}
{attribute 'TcGenerated'}
{attribute 'no-analysis'}
FUNCTION F_GetTitle : WSTRING
VAR_INPUT
	
END_VAR

F_GetTitle := "FsGenerics";

END_FUNCTION

// Project Information/F_GetVersion
// This function has been automatically generated from the project information.
{attribute 'signature_flag' := '1073741824'}
{attribute 'TcGenerated'}
{attribute 'no-analysis'}
FUNCTION F_GetVersion : ST_LibVersion
VAR_INPUT
	
END_VAR

F_GetVersion.iMajor := 0;
F_GetVersion.iMinor := 1;
F_GetVersion.iBuild := 1;
F_GetVersion.iRevision := 1;

END_FUNCTION
